TYPE ST_EL9410 :
STRUCT
	bit_UpUndervoltage	: BIT;
	bit_UsUndervoltage	: BIT;
	ui_state			: UINT;
END_STRUCT
END_TYPE

(* stored: Version 1.1.0.1, ProductVersion 3.1.4026.18
   DUT ST_EL9410: Id {7cd530dc-8d4c-4284-81c9-c21ec30607e1} *)
